PROGRAM Misalignments
VAR
END_VAR

//IF (Otto.PickupLocation1 OR Otto.PickupLocation2 OR Otto.PickupLocation3 OR
//	Otto.DropoffLocation1 OR Otto.DropoffLocation2 OR Otto.DropoffLocation3) AND Shuttle.Present = FALSE THEN
	
//	Supervisor.Misalignment := TRUE;
	
//ELSE
	
//	Supervisor.Misalignment := FALSE;

//END_IF

Supervisor.Misalignment := FALSE;

END_PROGRAM

(* stored: Version 1.1.0.1, ProductVersion 3.1.4024.9
   POU Misalignments: Id {c7c59819-1df4-4575-ba0e-0341bc2d34fb}, SpecialFunc None *)
